{attribute 'qualified_only'}
VAR_GLOBAL
	START : BOOL;
END_VAR

(* stored: Version 1.1.0.1, ProductVersion 3.1.4024.16
   GVL ROBOT: Id {6be28e65-6ea5-491d-a762-ca92440c5ee2} *)
